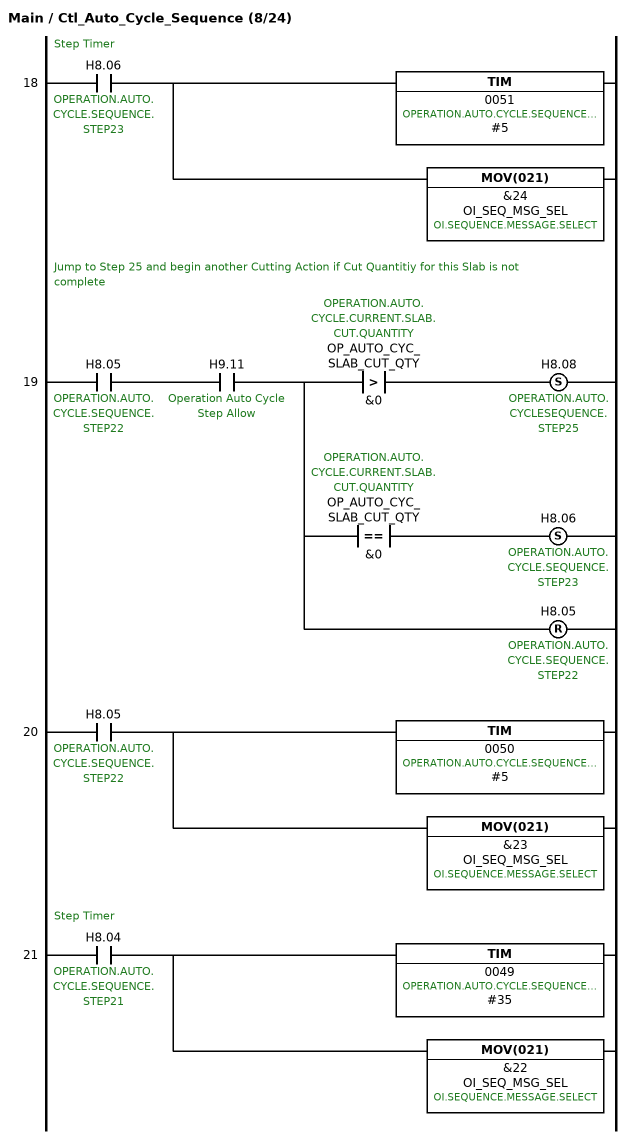
; [picture p24: Main / Ctl_Auto_Cycle_Sequence, rungs 18-21]
; rung 18: Step Timer
LD H8.06  ; OPERATION.AUTO.CYCLE.SEQUENCE.STEP23
TIM 0051 #5  ; OPERATION.AUTO.CYCLE.SEQUENCE.STEP23.TIMER
MOV(021) &24 OI_SEQ_MSG_SEL  ; OI.SEQUENCE.MESSAGE.SELECT
; rung 19: Jump to Step 25 and begin another Cutting Action if Cut Quantitiy for this Slab is not complete
LD H8.05  ; OPERATION.AUTO.CYCLE.SEQUENCE.STEP22
AND H9.11  ; Operation Auto Cycle Step Allow
OUT TR0
AND>(320) OP_AUTO_CYC_SLAB_CUT_QTY &0  ; OPERATION.AUTO.CYCLE.CURRENT.SLAB.CUT.QUANTITY
SET H8.08  ; OPERATION.AUTO.CYCLESEQUENCE.STEP25
LD TR0
AND=(300) OP_AUTO_CYC_SLAB_CUT_QTY &0  ; OPERATION.AUTO.CYCLE.CURRENT.SLAB.CUT.QUANTITY
SET H8.06  ; OPERATION.AUTO.CYCLE.SEQUENCE.STEP23
LD TR0
RSET H8.05  ; OPERATION.AUTO.CYCLE.SEQUENCE.STEP22
; rung 20
LD H8.05  ; OPERATION.AUTO.CYCLE.SEQUENCE.STEP22
TIM 0050 #5  ; OPERATION.AUTO.CYCLE.SEQUENCE.STEP22.TIMER
MOV(021) &23 OI_SEQ_MSG_SEL  ; OI.SEQUENCE.MESSAGE.SELECT
; rung 21: Step Timer
LD H8.04  ; OPERATION.AUTO.CYCLE.SEQUENCE.STEP21
TIM 0049 #35  ; OPERATION.AUTO.CYCLE.SEQUENCE.STEP21.TIMER
MOV(021) &22 OI_SEQ_MSG_SEL  ; OI.SEQUENCE.MESSAGE.SELECT

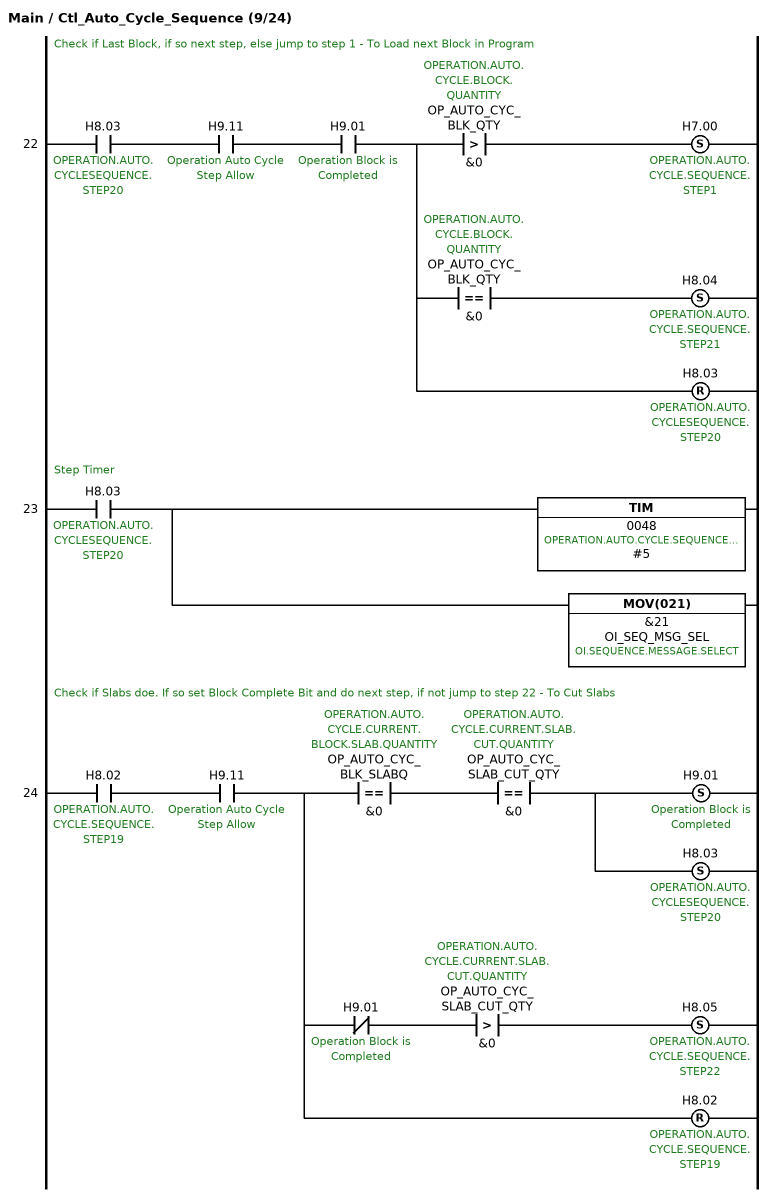
; rung 22: Check if Last Block, if so next step, else jump to step 1 - To Load next Block in Program
LD H8.03  ; OPERATION.AUTO.CYCLESEQUENCE.STEP20
AND H9.11  ; Operation Auto Cycle Step Allow
AND H9.01  ; Operation Block is Completed
OUT TR0
AND>(320) OP_AUTO_CYC_BLK_QTY &0  ; OPERATION.AUTO.CYCLE.BLOCK.QUANTITY
SET H7.00  ; OPERATION.AUTO.CYCLE.SEQUENCE.STEP1
LD TR0
AND=(300) OP_AUTO_CYC_BLK_QTY &0  ; OPERATION.AUTO.CYCLE.BLOCK.QUANTITY
SET H8.04  ; OPERATION.AUTO.CYCLE.SEQUENCE.STEP21
LD TR0
RSET H8.03  ; OPERATION.AUTO.CYCLESEQUENCE.STEP20
; rung 23: Step Timer
LD H8.03  ; OPERATION.AUTO.CYCLESEQUENCE.STEP20
TIM 0048 #5  ; OPERATION.AUTO.CYCLE.SEQUENCE.STEP20.TIMER
MOV(021) &21 OI_SEQ_MSG_SEL  ; OI.SEQUENCE.MESSAGE.SELECT
; rung 24: Check if Slabs doe. If so set Block Complete Bit and do next step, if not jump to step 22 - To Cut Slabs
LD H8.02  ; OPERATION.AUTO.CYCLE.SEQUENCE.STEP19
AND H9.11  ; Operation Auto Cycle Step Allow
OUT TR0
AND=(300) OP_AUTO_CYC_BLK_SLABQ &0  ; OPERATION.AUTO.CYCLE.CURRENT.BLOCK.SLAB.QUANTITY
AND=(300) OP_AUTO_CYC_SLAB_CUT_QTY &0  ; OPERATION.AUTO.CYCLE.CURRENT.SLAB.CUT.QUANTITY
SET H9.01  ; Operation Block is Completed
SET H8.03  ; OPERATION.AUTO.CYCLESEQUENCE.STEP20
LD TR0
ANDNOT H9.01  ; Operation Block is Completed
AND>(320) OP_AUTO_CYC_SLAB_CUT_QTY &0  ; OPERATION.AUTO.CYCLE.CURRENT.SLAB.CUT.QUANTITY
SET H8.05  ; OPERATION.AUTO.CYCLE.SEQUENCE.STEP22
LD TR0
RSET H8.02  ; OPERATION.AUTO.CYCLE.SEQUENCE.STEP19

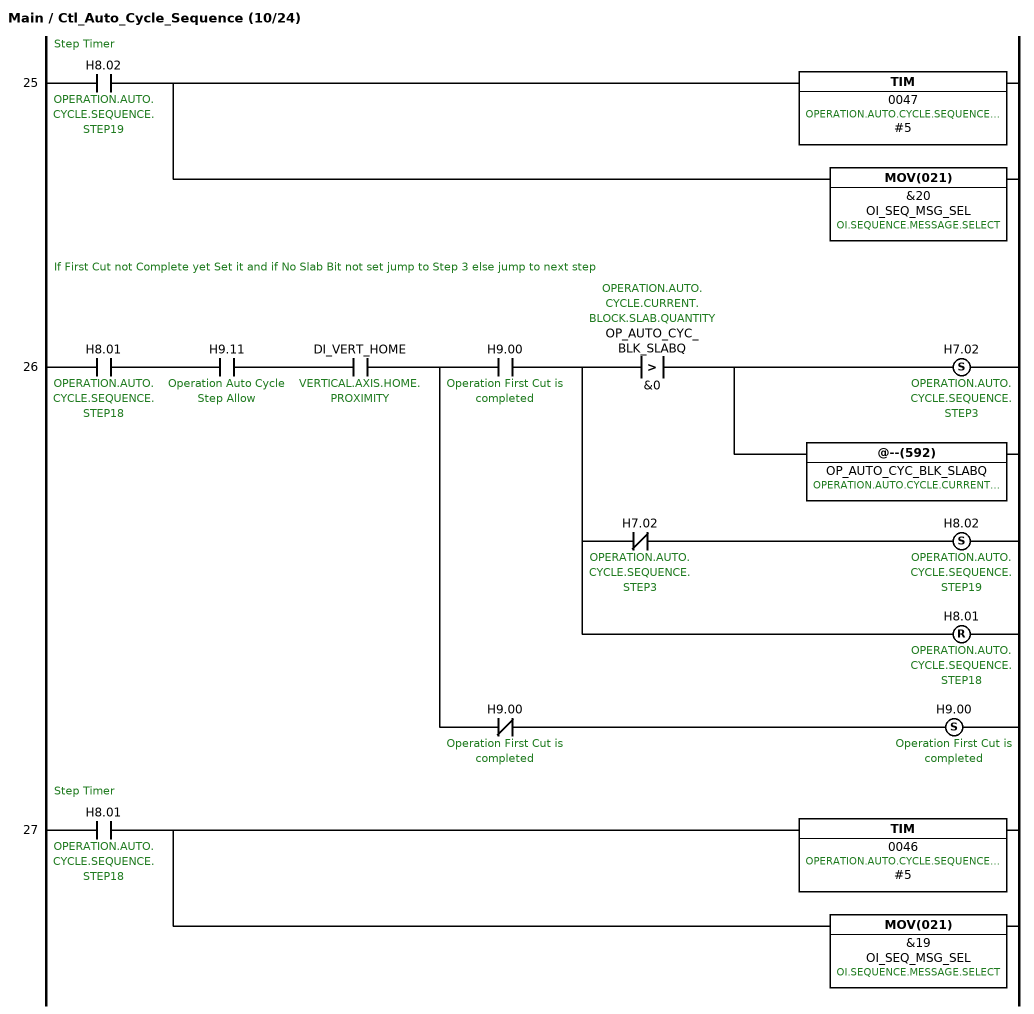
; rung 25: Step Timer
LD H8.02  ; OPERATION.AUTO.CYCLE.SEQUENCE.STEP19
TIM 0047 #5  ; OPERATION.AUTO.CYCLE.SEQUENCE.STEP19.TIMER
MOV(021) &20 OI_SEQ_MSG_SEL  ; OI.SEQUENCE.MESSAGE.SELECT
; rung 26: If First Cut not Complete yet Set it and if No Slab Bit not set jump to Step 3 else jump to next step
LD H8.01  ; OPERATION.AUTO.CYCLE.SEQUENCE.STEP18
AND H9.11  ; Operation Auto Cycle Step Allow
AND DI_VERT_HOME  ; VERTICAL.AXIS.HOME.PROXIMITY
OUT TR0
AND H9.00  ; Operation First Cut is completed
OUT TR1
AND>(320) OP_AUTO_CYC_BLK_SLABQ &0  ; OPERATION.AUTO.CYCLE.CURRENT.BLOCK.SLAB.QUANTITY
SET H7.02  ; OPERATION.AUTO.CYCLE.SEQUENCE.STEP3
@--(592) OP_AUTO_CYC_BLK_SLABQ  ; OPERATION.AUTO.CYCLE.CURRENT.BLOCK.SLAB.QUANTITY
LD TR1
ANDNOT H7.02  ; OPERATION.AUTO.CYCLE.SEQUENCE.STEP3
SET H8.02  ; OPERATION.AUTO.CYCLE.SEQUENCE.STEP19
LD TR1
RSET H8.01  ; OPERATION.AUTO.CYCLE.SEQUENCE.STEP18
LD TR0
ANDNOT H9.00  ; Operation First Cut is completed
SET H9.00  ; Operation First Cut is completed
; rung 27: Step Timer
LD H8.01  ; OPERATION.AUTO.CYCLE.SEQUENCE.STEP18
TIM 0046 #5  ; OPERATION.AUTO.CYCLE.SEQUENCE.STEP18.TIMER
MOV(021) &19 OI_SEQ_MSG_SEL  ; OI.SEQUENCE.MESSAGE.SELECT

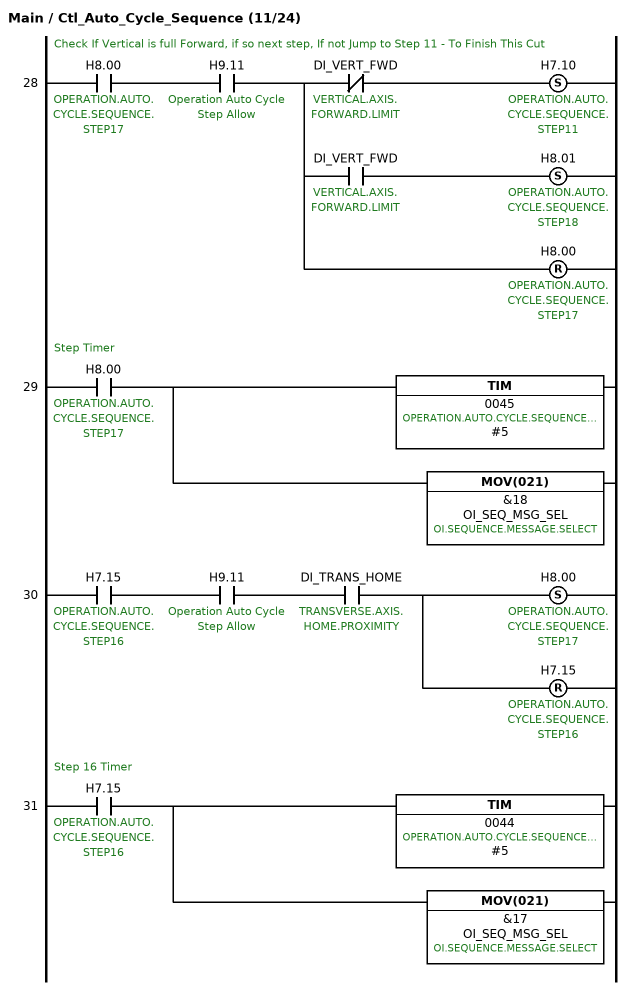
; rung 28: Check If Vertical is full Forward, if so next step, If not Jump to Step 11 - To Finish This Cut
LD H8.00  ; OPERATION.AUTO.CYCLE.SEQUENCE.STEP17
AND H9.11  ; Operation Auto Cycle Step Allow
OUT TR0
ANDNOT DI_VERT_FWD  ; VERTICAL.AXIS.FORWARD.LIMIT
SET H7.10  ; OPERATION.AUTO.CYCLE.SEQUENCE.STEP11
LD TR0
AND DI_VERT_FWD  ; VERTICAL.AXIS.FORWARD.LIMIT
SET H8.01  ; OPERATION.AUTO.CYCLE.SEQUENCE.STEP18
LD TR0
RSET H8.00  ; OPERATION.AUTO.CYCLE.SEQUENCE.STEP17
; rung 29: Step Timer
LD H8.00  ; OPERATION.AUTO.CYCLE.SEQUENCE.STEP17
TIM 0045 #5  ; OPERATION.AUTO.CYCLE.SEQUENCE.STEP17.TIMER
MOV(021) &18 OI_SEQ_MSG_SEL  ; OI.SEQUENCE.MESSAGE.SELECT
; rung 30
LD H7.15  ; OPERATION.AUTO.CYCLE.SEQUENCE.STEP16
AND H9.11  ; Operation Auto Cycle Step Allow
AND DI_TRANS_HOME  ; TRANSVERSE.AXIS.HOME.PROXIMITY
SET H8.00  ; OPERATION.AUTO.CYCLE.SEQUENCE.STEP17
RSET H7.15  ; OPERATION.AUTO.CYCLE.SEQUENCE.STEP16
; rung 31: Step 16 Timer
LD H7.15  ; OPERATION.AUTO.CYCLE.SEQUENCE.STEP16
TIM 0044 #5  ; OPERATION.AUTO.CYCLE.SEQUENCE.STEP16.TIMER
MOV(021) &17 OI_SEQ_MSG_SEL  ; OI.SEQUENCE.MESSAGE.SELECT

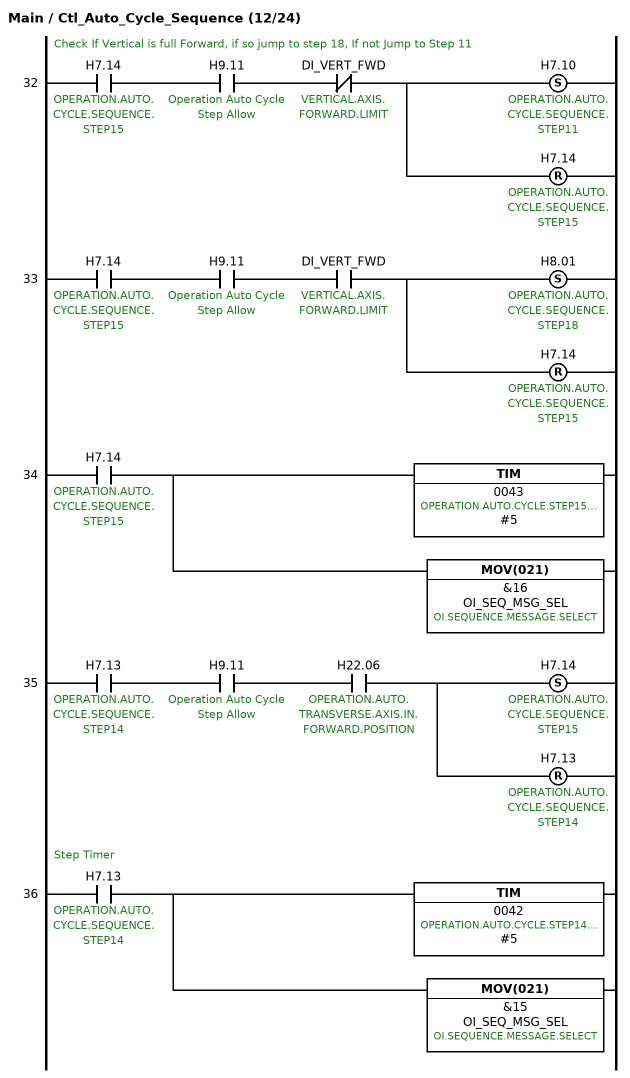
; rung 32: Check If Vertical is full Forward, if so jump to step 18, If not Jump to Step 11
LD H7.14  ; OPERATION.AUTO.CYCLE.SEQUENCE.STEP15
AND H9.11  ; Operation Auto Cycle Step Allow
ANDNOT DI_VERT_FWD  ; VERTICAL.AXIS.FORWARD.LIMIT
SET H7.10  ; OPERATION.AUTO.CYCLE.SEQUENCE.STEP11
RSET H7.14  ; OPERATION.AUTO.CYCLE.SEQUENCE.STEP15
; rung 33
LD H7.14  ; OPERATION.AUTO.CYCLE.SEQUENCE.STEP15
AND H9.11  ; Operation Auto Cycle Step Allow
AND DI_VERT_FWD  ; VERTICAL.AXIS.FORWARD.LIMIT
SET H8.01  ; OPERATION.AUTO.CYCLE.SEQUENCE.STEP18
RSET H7.14  ; OPERATION.AUTO.CYCLE.SEQUENCE.STEP15
; rung 34
LD H7.14  ; OPERATION.AUTO.CYCLE.SEQUENCE.STEP15
TIM 0043 #5  ; OPERATION.AUTO.CYCLE.STEP15.TIMER
MOV(021) &16 OI_SEQ_MSG_SEL  ; OI.SEQUENCE.MESSAGE.SELECT
; rung 35
LD H7.13  ; OPERATION.AUTO.CYCLE.SEQUENCE.STEP14
AND H9.11  ; Operation Auto Cycle Step Allow
AND H22.06  ; OPERATION.AUTO.TRANSVERSE.AXIS.IN.FORWARD.POSITION
SET H7.14  ; OPERATION.AUTO.CYCLE.SEQUENCE.STEP15
RSET H7.13  ; OPERATION.AUTO.CYCLE.SEQUENCE.STEP14
; rung 36: Step Timer
LD H7.13  ; OPERATION.AUTO.CYCLE.SEQUENCE.STEP14
TIM 0042 #5  ; OPERATION.AUTO.CYCLE.STEP14.TIMER
MOV(021) &15 OI_SEQ_MSG_SEL  ; OI.SEQUENCE.MESSAGE.SELECT

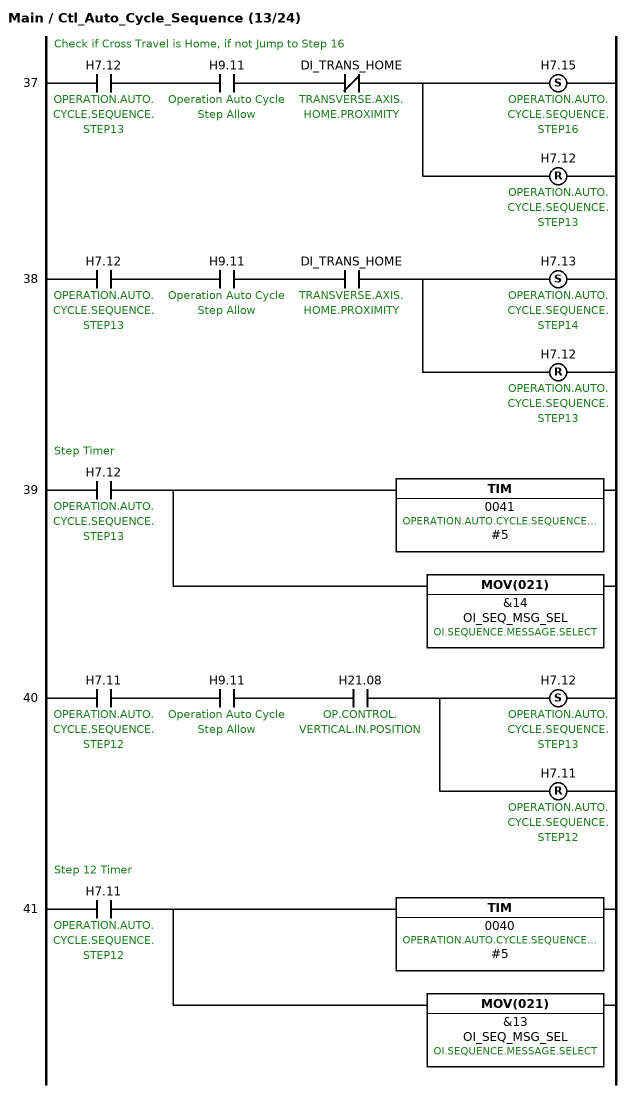
; rung 37: Check if Cross Travel is Home, if not Jump to Step 16
LD H7.12  ; OPERATION.AUTO.CYCLE.SEQUENCE.STEP13
AND H9.11  ; Operation Auto Cycle Step Allow
ANDNOT DI_TRANS_HOME  ; TRANSVERSE.AXIS.HOME.PROXIMITY
SET H7.15  ; OPERATION.AUTO.CYCLE.SEQUENCE.STEP16
RSET H7.12  ; OPERATION.AUTO.CYCLE.SEQUENCE.STEP13
; rung 38
LD H7.12  ; OPERATION.AUTO.CYCLE.SEQUENCE.STEP13
AND H9.11  ; Operation Auto Cycle Step Allow
AND DI_TRANS_HOME  ; TRANSVERSE.AXIS.HOME.PROXIMITY
SET H7.13  ; OPERATION.AUTO.CYCLE.SEQUENCE.STEP14
RSET H7.12  ; OPERATION.AUTO.CYCLE.SEQUENCE.STEP13
; rung 39: Step Timer
LD H7.12  ; OPERATION.AUTO.CYCLE.SEQUENCE.STEP13
TIM 0041 #5  ; OPERATION.AUTO.CYCLE.SEQUENCE.STEP13.TIME
MOV(021) &14 OI_SEQ_MSG_SEL  ; OI.SEQUENCE.MESSAGE.SELECT
; rung 40
LD H7.11  ; OPERATION.AUTO.CYCLE.SEQUENCE.STEP12
AND H9.11  ; Operation Auto Cycle Step Allow
AND H21.08  ; OP.CONTROL.VERTICAL.IN.POSITION
SET H7.12  ; OPERATION.AUTO.CYCLE.SEQUENCE.STEP13
RSET H7.11  ; OPERATION.AUTO.CYCLE.SEQUENCE.STEP12
; rung 41: Step 12 Timer
LD H7.11  ; OPERATION.AUTO.CYCLE.SEQUENCE.STEP12
TIM 0040 #5  ; OPERATION.AUTO.CYCLE.SEQUENCE.STEP12.TIMER
MOV(021) &13 OI_SEQ_MSG_SEL  ; OI.SEQUENCE.MESSAGE.SELECT

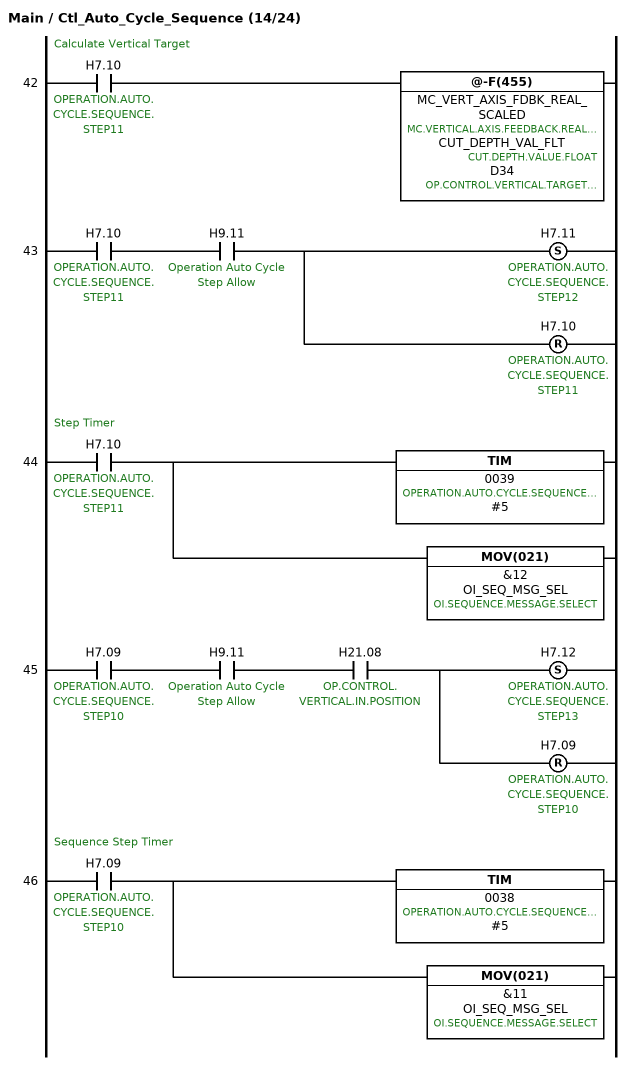
; rung 42: Calculate Vertical Target
LD H7.10  ; OPERATION.AUTO.CYCLE.SEQUENCE.STEP11
@-F(455) MC_VERT_AXIS_FDBK_REAL_SCALED CUT_DEPTH_VAL_FLT D34  ; MC.VERTICAL.AXIS.FEEDBACK.REAL.SCALED.INCH, CUT.DEPTH.VALUE.FLOAT, OP.CONTROL.VERTICAL.TARGET.SCALED
; rung 43
LD H7.10  ; OPERATION.AUTO.CYCLE.SEQUENCE.STEP11
AND H9.11  ; Operation Auto Cycle Step Allow
SET H7.11  ; OPERATION.AUTO.CYCLE.SEQUENCE.STEP12
RSET H7.10  ; OPERATION.AUTO.CYCLE.SEQUENCE.STEP11
; rung 44: Step Timer
LD H7.10  ; OPERATION.AUTO.CYCLE.SEQUENCE.STEP11
TIM 0039 #5  ; OPERATION.AUTO.CYCLE.SEQUENCE.STEP11.TIMER
MOV(021) &12 OI_SEQ_MSG_SEL  ; OI.SEQUENCE.MESSAGE.SELECT
; rung 45
LD H7.09  ; OPERATION.AUTO.CYCLE.SEQUENCE.STEP10
AND H9.11  ; Operation Auto Cycle Step Allow
AND H21.08  ; OP.CONTROL.VERTICAL.IN.POSITION
SET H7.12  ; OPERATION.AUTO.CYCLE.SEQUENCE.STEP13
RSET H7.09  ; OPERATION.AUTO.CYCLE.SEQUENCE.STEP10
; rung 46: Sequence Step Timer
LD H7.09  ; OPERATION.AUTO.CYCLE.SEQUENCE.STEP10
TIM 0038 #5  ; OPERATION.AUTO.CYCLE.SEQUENCE.STEP10.TIMER
MOV(021) &11 OI_SEQ_MSG_SEL  ; OI.SEQUENCE.MESSAGE.SELECT

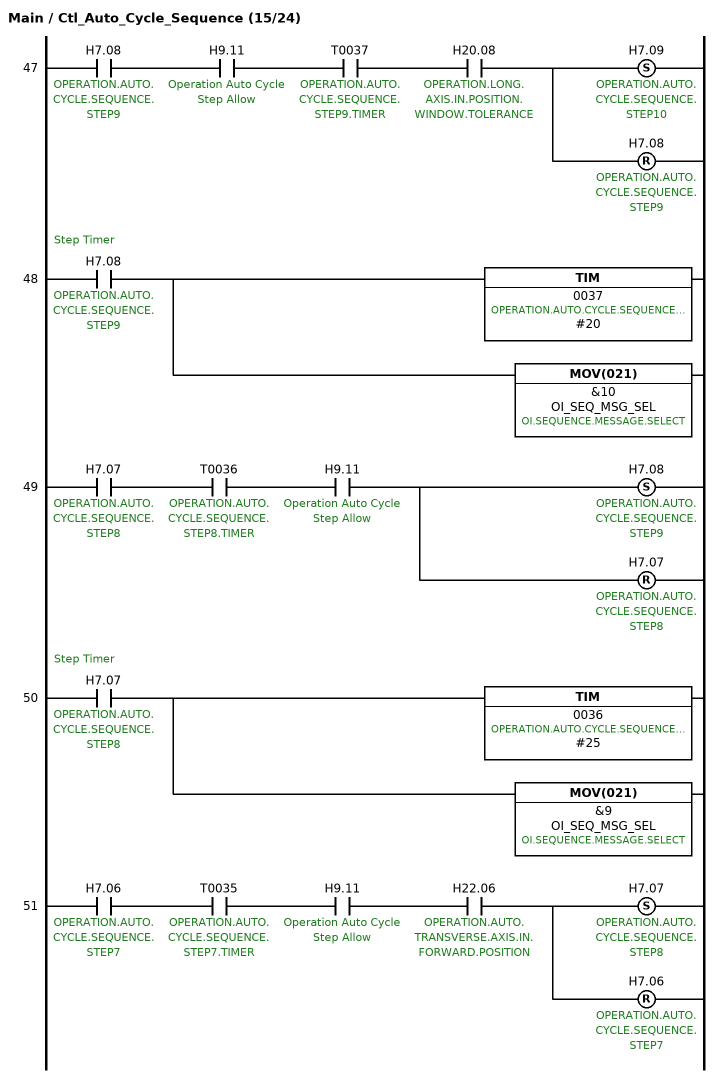
; rung 47
LD H7.08  ; OPERATION.AUTO.CYCLE.SEQUENCE.STEP9
AND H9.11  ; Operation Auto Cycle Step Allow
AND T0037  ; OPERATION.AUTO.CYCLE.SEQUENCE.STEP9.TIMER
AND H20.08  ; OPERATION.LONG.AXIS.IN.POSITION.WINDOW.TOLERANCE
SET H7.09  ; OPERATION.AUTO.CYCLE.SEQUENCE.STEP10
RSET H7.08  ; OPERATION.AUTO.CYCLE.SEQUENCE.STEP9
; rung 48: Step Timer
LD H7.08  ; OPERATION.AUTO.CYCLE.SEQUENCE.STEP9
TIM 0037 #20  ; OPERATION.AUTO.CYCLE.SEQUENCE.STEP9.TIMER
MOV(021) &10 OI_SEQ_MSG_SEL  ; OI.SEQUENCE.MESSAGE.SELECT
; rung 49
LD H7.07  ; OPERATION.AUTO.CYCLE.SEQUENCE.STEP8
AND T0036  ; OPERATION.AUTO.CYCLE.SEQUENCE.STEP8.TIMER
AND H9.11  ; Operation Auto Cycle Step Allow
SET H7.08  ; OPERATION.AUTO.CYCLE.SEQUENCE.STEP9
RSET H7.07  ; OPERATION.AUTO.CYCLE.SEQUENCE.STEP8
; rung 50: Step Timer
LD H7.07  ; OPERATION.AUTO.CYCLE.SEQUENCE.STEP8
TIM 0036 #25  ; OPERATION.AUTO.CYCLE.SEQUENCE.STEP8.TIMER
MOV(021) &9 OI_SEQ_MSG_SEL  ; OI.SEQUENCE.MESSAGE.SELECT
; rung 51
LD H7.06  ; OPERATION.AUTO.CYCLE.SEQUENCE.STEP7
AND T0035  ; OPERATION.AUTO.CYCLE.SEQUENCE.STEP7.TIMER
AND H9.11  ; Operation Auto Cycle Step Allow
AND H22.06  ; OPERATION.AUTO.TRANSVERSE.AXIS.IN.FORWARD.POSITION
SET H7.07  ; OPERATION.AUTO.CYCLE.SEQUENCE.STEP8
RSET H7.06  ; OPERATION.AUTO.CYCLE.SEQUENCE.STEP7

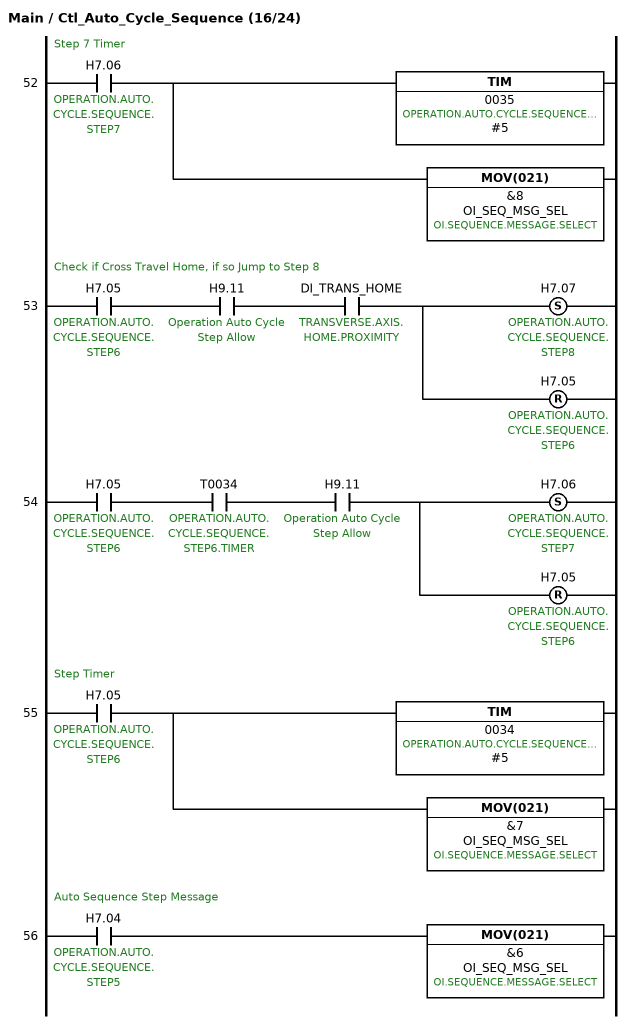
; rung 52: Step 7 Timer
LD H7.06  ; OPERATION.AUTO.CYCLE.SEQUENCE.STEP7
TIM 0035 #5  ; OPERATION.AUTO.CYCLE.SEQUENCE.STEP7.TIMER
MOV(021) &8 OI_SEQ_MSG_SEL  ; OI.SEQUENCE.MESSAGE.SELECT
; rung 53: Check if Cross Travel Home, if so Jump to Step 8
LD H7.05  ; OPERATION.AUTO.CYCLE.SEQUENCE.STEP6
AND H9.11  ; Operation Auto Cycle Step Allow
AND DI_TRANS_HOME  ; TRANSVERSE.AXIS.HOME.PROXIMITY
SET H7.07  ; OPERATION.AUTO.CYCLE.SEQUENCE.STEP8
RSET H7.05  ; OPERATION.AUTO.CYCLE.SEQUENCE.STEP6
; rung 54
LD H7.05  ; OPERATION.AUTO.CYCLE.SEQUENCE.STEP6
AND T0034  ; OPERATION.AUTO.CYCLE.SEQUENCE.STEP6.TIMER
AND H9.11  ; Operation Auto Cycle Step Allow
SET H7.06  ; OPERATION.AUTO.CYCLE.SEQUENCE.STEP7
RSET H7.05  ; OPERATION.AUTO.CYCLE.SEQUENCE.STEP6
; rung 55: Step Timer
LD H7.05  ; OPERATION.AUTO.CYCLE.SEQUENCE.STEP6
TIM 0034 #5  ; OPERATION.AUTO.CYCLE.SEQUENCE.STEP6.TIMER
MOV(021) &7 OI_SEQ_MSG_SEL  ; OI.SEQUENCE.MESSAGE.SELECT
; rung 56: Auto Sequence Step Message
LD H7.04  ; OPERATION.AUTO.CYCLE.SEQUENCE.STEP5
MOV(021) &6 OI_SEQ_MSG_SEL  ; OI.SEQUENCE.MESSAGE.SELECT

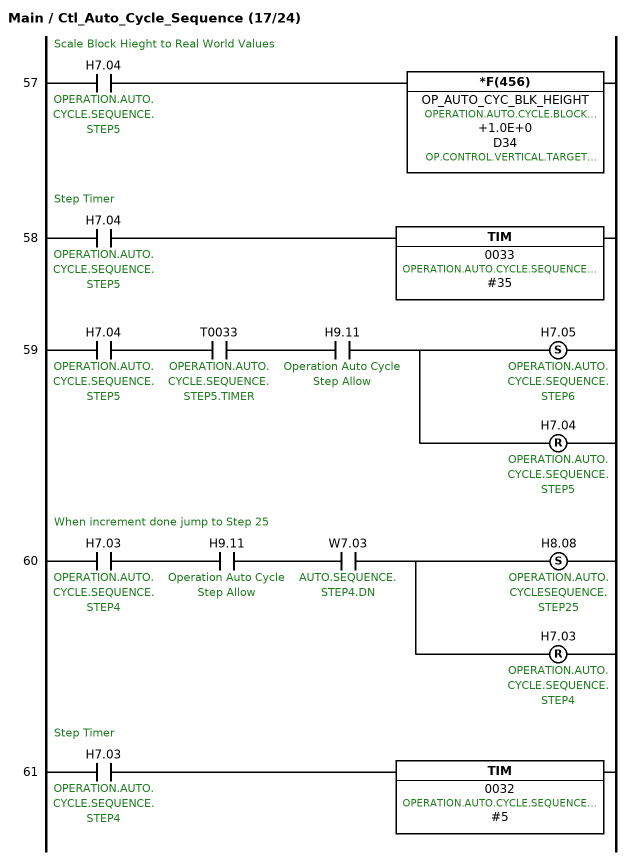
; rung 57: Scale Block Hieght to Real World Values
LD H7.04  ; OPERATION.AUTO.CYCLE.SEQUENCE.STEP5
*F(456) OP_AUTO_CYC_BLK_HEIGHT +1.0E+0 D34  ; OPERATION.AUTO.CYCLE.BLOCK.HEIGHT.WORKING, OP.CONTROL.VERTICAL.TARGET.SCALED
; rung 58: Step Timer
LD H7.04  ; OPERATION.AUTO.CYCLE.SEQUENCE.STEP5
TIM 0033 #35  ; OPERATION.AUTO.CYCLE.SEQUENCE.STEP5.TIMER
; rung 59
LD H7.04  ; OPERATION.AUTO.CYCLE.SEQUENCE.STEP5
AND T0033  ; OPERATION.AUTO.CYCLE.SEQUENCE.STEP5.TIMER
AND H9.11  ; Operation Auto Cycle Step Allow
SET H7.05  ; OPERATION.AUTO.CYCLE.SEQUENCE.STEP6
RSET H7.04  ; OPERATION.AUTO.CYCLE.SEQUENCE.STEP5
; rung 60: When increment done jump to Step 25
LD H7.03  ; OPERATION.AUTO.CYCLE.SEQUENCE.STEP4
AND H9.11  ; Operation Auto Cycle Step Allow
AND W7.03  ; AUTO.SEQUENCE.STEP4.DN
SET H8.08  ; OPERATION.AUTO.CYCLESEQUENCE.STEP25
RSET H7.03  ; OPERATION.AUTO.CYCLE.SEQUENCE.STEP4
; rung 61: Step Timer
LD H7.03  ; OPERATION.AUTO.CYCLE.SEQUENCE.STEP4
TIM 0032 #5  ; OPERATION.AUTO.CYCLE.SEQUENCE.STEP4.TIMER

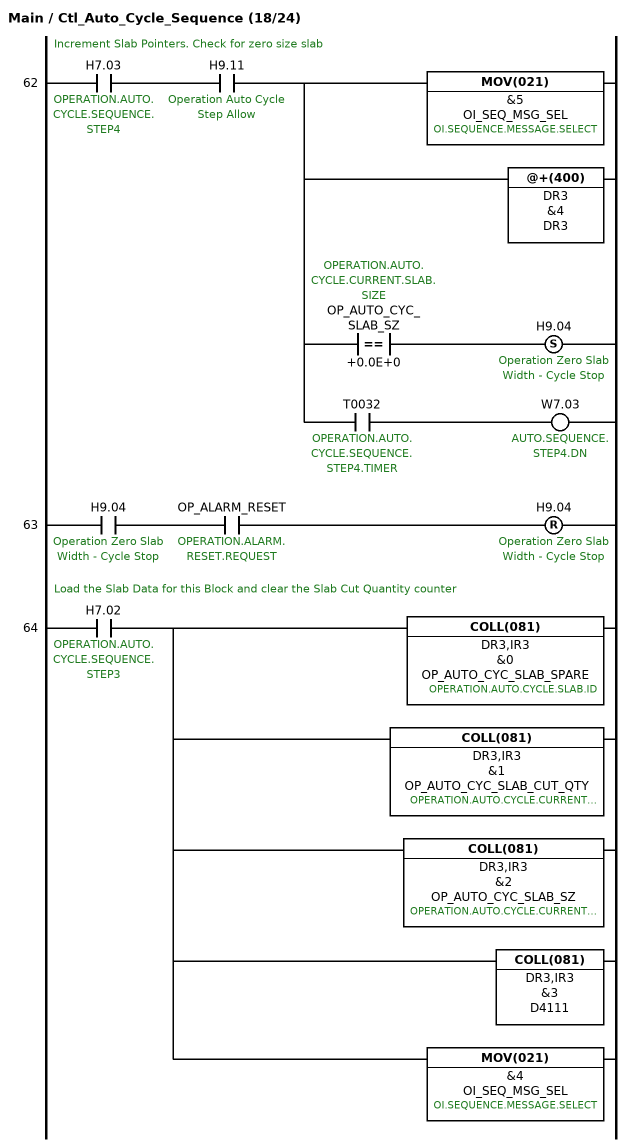
; rung 62: Increment Slab Pointers. Check for zero size slab
LD H7.03  ; OPERATION.AUTO.CYCLE.SEQUENCE.STEP4
AND H9.11  ; Operation Auto Cycle Step Allow
OUT TR0
MOV(021) &5 OI_SEQ_MSG_SEL  ; OI.SEQUENCE.MESSAGE.SELECT
@+(400) DR3 &4 DR3
AND=F(329) OP_AUTO_CYC_SLAB_SZ +0.0E+0  ; OPERATION.AUTO.CYCLE.CURRENT.SLAB.SIZE
SET H9.04  ; Operation Zero Slab Width - Cycle Stop
LD TR0
AND T0032  ; OPERATION.AUTO.CYCLE.SEQUENCE.STEP4.TIMER
OUT W7.03  ; AUTO.SEQUENCE.STEP4.DN
; rung 63
LD H9.04  ; Operation Zero Slab Width - Cycle Stop
AND OP_ALARM_RESET  ; OPERATION.ALARM.RESET.REQUEST
RSET H9.04  ; Operation Zero Slab Width - Cycle Stop
; rung 64: Load the Slab Data for this Block and clear the Slab Cut Quantity counter
LD H7.02  ; OPERATION.AUTO.CYCLE.SEQUENCE.STEP3
COLL(081) DR3,IR3 &0 OP_AUTO_CYC_SLAB_SPARE  ; OPERATION.AUTO.CYCLE.SLAB.ID
COLL(081) DR3,IR3 &1 OP_AUTO_CYC_SLAB_CUT_QTY  ; OPERATION.AUTO.CYCLE.CURRENT.SLAB.CUT.QUANTITY
COLL(081) DR3,IR3 &2 OP_AUTO_CYC_SLAB_SZ  ; OPERATION.AUTO.CYCLE.CURRENT.SLAB.SIZE
COLL(081) DR3,IR3 &3 D4111
MOV(021) &4 OI_SEQ_MSG_SEL  ; OI.SEQUENCE.MESSAGE.SELECT

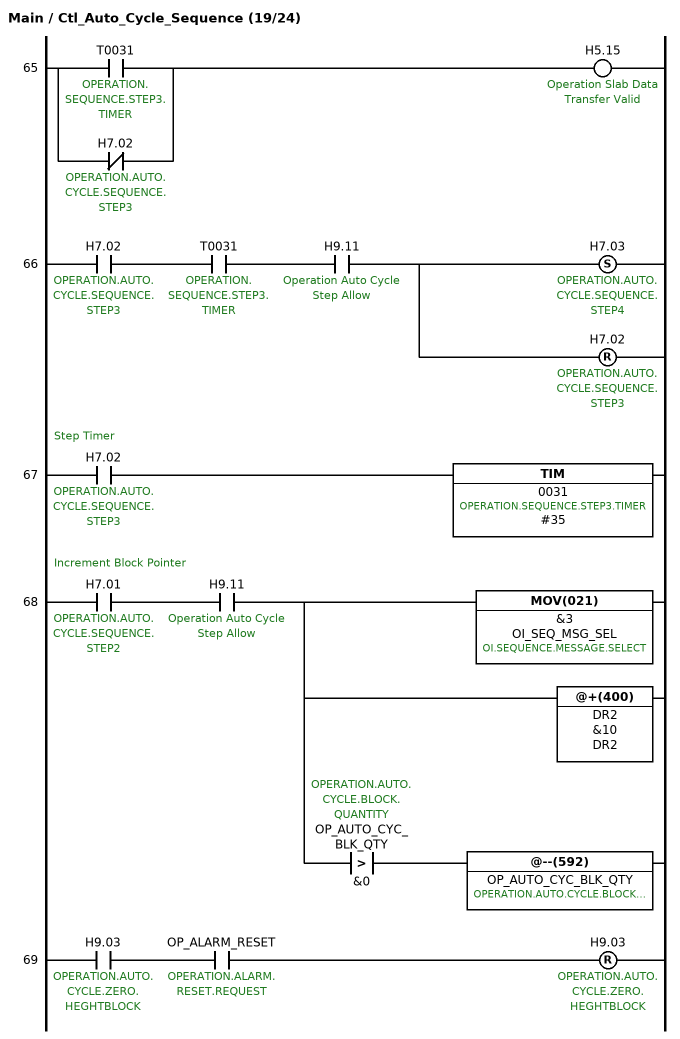
; rung 65
LD T0031  ; OPERATION.SEQUENCE.STEP3.TIMER
ORNOT H7.02  ; OPERATION.AUTO.CYCLE.SEQUENCE.STEP3
OUT H5.15  ; Operation Slab Data Transfer Valid
; rung 66
LD H7.02  ; OPERATION.AUTO.CYCLE.SEQUENCE.STEP3
AND T0031  ; OPERATION.SEQUENCE.STEP3.TIMER
AND H9.11  ; Operation Auto Cycle Step Allow
SET H7.03  ; OPERATION.AUTO.CYCLE.SEQUENCE.STEP4
RSET H7.02  ; OPERATION.AUTO.CYCLE.SEQUENCE.STEP3
; rung 67: Step Timer
LD H7.02  ; OPERATION.AUTO.CYCLE.SEQUENCE.STEP3
TIM 0031 #35  ; OPERATION.SEQUENCE.STEP3.TIMER
; rung 68: Increment Block Pointer
LD H7.01  ; OPERATION.AUTO.CYCLE.SEQUENCE.STEP2
AND H9.11  ; Operation Auto Cycle Step Allow
MOV(021) &3 OI_SEQ_MSG_SEL  ; OI.SEQUENCE.MESSAGE.SELECT
@+(400) DR2 &10 DR2
AND>(320) OP_AUTO_CYC_BLK_QTY &0  ; OPERATION.AUTO.CYCLE.BLOCK.QUANTITY
@--(592) OP_AUTO_CYC_BLK_QTY  ; OPERATION.AUTO.CYCLE.BLOCK.QUANTITY
; rung 69
LD H9.03  ; OPERATION.AUTO.CYCLE.ZERO.HEGHTBLOCK
AND OP_ALARM_RESET  ; OPERATION.ALARM.RESET.REQUEST
RSET H9.03  ; OPERATION.AUTO.CYCLE.ZERO.HEGHTBLOCK

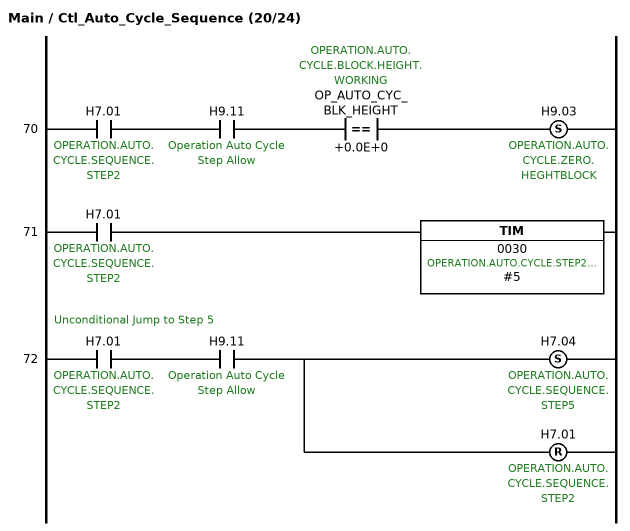
; rung 70
LD H7.01  ; OPERATION.AUTO.CYCLE.SEQUENCE.STEP2
AND H9.11  ; Operation Auto Cycle Step Allow
AND=F(329) OP_AUTO_CYC_BLK_HEIGHT +0.0E+0  ; OPERATION.AUTO.CYCLE.BLOCK.HEIGHT.WORKING
SET H9.03  ; OPERATION.AUTO.CYCLE.ZERO.HEGHTBLOCK
; rung 71
LD H7.01  ; OPERATION.AUTO.CYCLE.SEQUENCE.STEP2
TIM 0030 #5  ; OPERATION.AUTO.CYCLE.STEP2.TIMER
; rung 72: Unconditional Jump to Step 5
LD H7.01  ; OPERATION.AUTO.CYCLE.SEQUENCE.STEP2
AND H9.11  ; Operation Auto Cycle Step Allow
SET H7.04  ; OPERATION.AUTO.CYCLE.SEQUENCE.STEP5
RSET H7.01  ; OPERATION.AUTO.CYCLE.SEQUENCE.STEP2

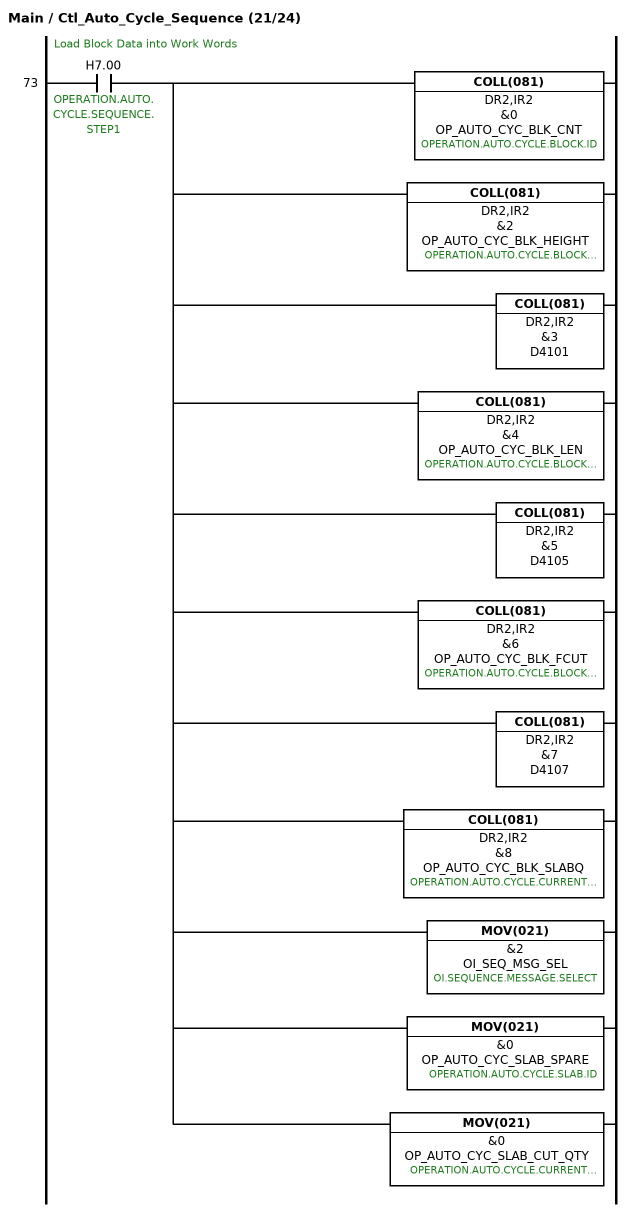
; rung 73: Load Block Data into Work Words
LD H7.00  ; OPERATION.AUTO.CYCLE.SEQUENCE.STEP1
COLL(081) DR2,IR2 &0 OP_AUTO_CYC_BLK_CNT  ; OPERATION.AUTO.CYCLE.BLOCK.ID
COLL(081) DR2,IR2 &2 OP_AUTO_CYC_BLK_HEIGHT  ; OPERATION.AUTO.CYCLE.BLOCK.HEIGHT.WORKING
COLL(081) DR2,IR2 &3 D4101
COLL(081) DR2,IR2 &4 OP_AUTO_CYC_BLK_LEN  ; OPERATION.AUTO.CYCLE.BLOCK.TRANSVERSE.AXIS.STOP.POSITION.WORKING
COLL(081) DR2,IR2 &5 D4105
COLL(081) DR2,IR2 &6 OP_AUTO_CYC_BLK_FCUT  ; OPERATION.AUTO.CYCLE.BLOCK.FIRST.CUT.WORKING
COLL(081) DR2,IR2 &7 D4107
COLL(081) DR2,IR2 &8 OP_AUTO_CYC_BLK_SLABQ  ; OPERATION.AUTO.CYCLE.CURRENT.BLOCK.SLAB.QUANTITY
MOV(021) &2 OI_SEQ_MSG_SEL  ; OI.SEQUENCE.MESSAGE.SELECT
MOV(021) &0 OP_AUTO_CYC_SLAB_SPARE  ; OPERATION.AUTO.CYCLE.SLAB.ID
MOV(021) &0 OP_AUTO_CYC_SLAB_CUT_QTY  ; OPERATION.AUTO.CYCLE.CURRENT.SLAB.CUT.QUANTITY

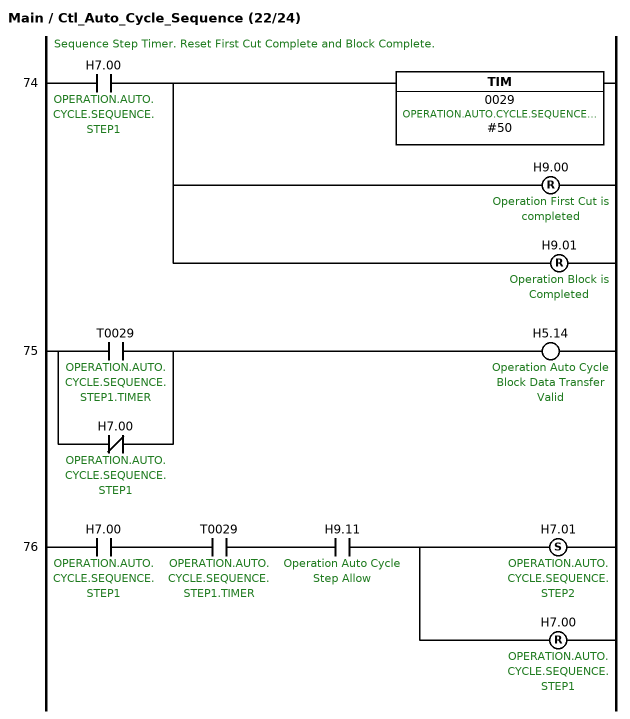
; rung 74: Sequence Step Timer. Reset First Cut Complete and Block Complete.
LD H7.00  ; OPERATION.AUTO.CYCLE.SEQUENCE.STEP1
TIM 0029 #50  ; OPERATION.AUTO.CYCLE.SEQUENCE.STEP1.TIMER
RSET H9.00  ; Operation First Cut is completed
RSET H9.01  ; Operation Block is Completed
; rung 75
LD T0029  ; OPERATION.AUTO.CYCLE.SEQUENCE.STEP1.TIMER
ORNOT H7.00  ; OPERATION.AUTO.CYCLE.SEQUENCE.STEP1
OUT H5.14  ; Operation Auto Cycle Block Data Transfer Valid
; rung 76
LD H7.00  ; OPERATION.AUTO.CYCLE.SEQUENCE.STEP1
AND T0029  ; OPERATION.AUTO.CYCLE.SEQUENCE.STEP1.TIMER
AND H9.11  ; Operation Auto Cycle Step Allow
SET H7.01  ; OPERATION.AUTO.CYCLE.SEQUENCE.STEP2
RSET H7.00  ; OPERATION.AUTO.CYCLE.SEQUENCE.STEP1

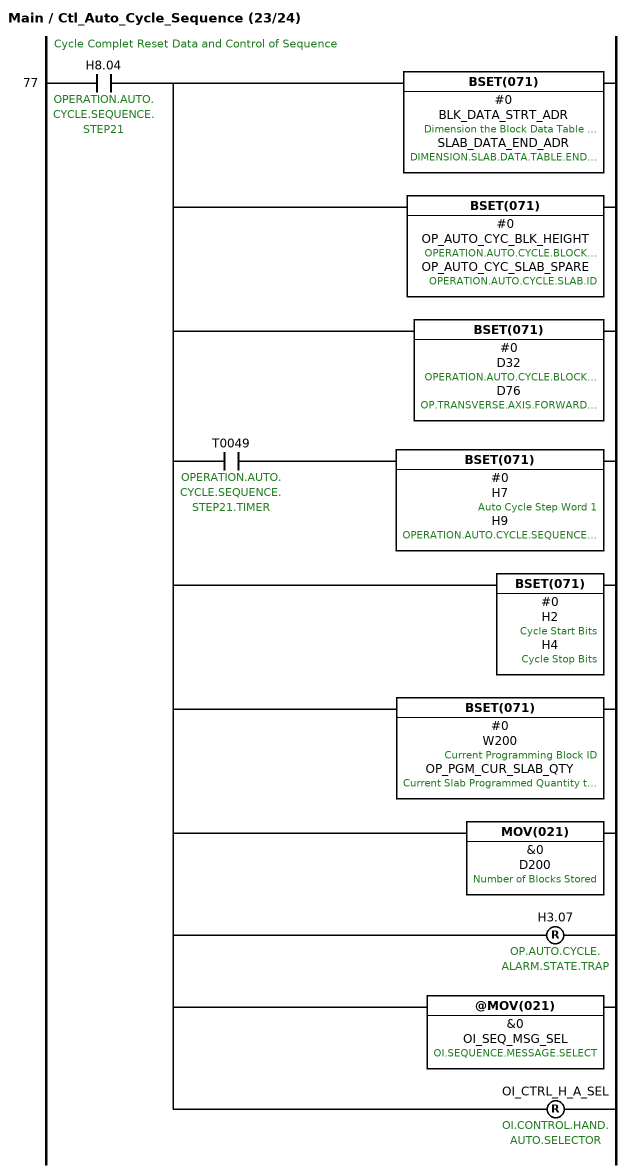
; rung 77: Cycle Complet Reset Data and Control of Sequence
LD H8.04  ; OPERATION.AUTO.CYCLE.SEQUENCE.STEP21
OUT TR0
BSET(071) #0 BLK_DATA_STRT_ADR SLAB_DATA_END_ADR  ; Dimension the Block Data Table - Start Address, DIMENSION.SLAB.DATA.TABLE.END.ADDRESS
BSET(071) #0 OP_AUTO_CYC_BLK_HEIGHT OP_AUTO_CYC_SLAB_SPARE  ; OPERATION.AUTO.CYCLE.BLOCK.HEIGHT.WORKING, OPERATION.AUTO.CYCLE.SLAB.ID
BSET(071) #0 D32 D76  ; OPERATION.AUTO.CYCLE.BLOCK.FIRST.CUT.WORKING.REAL, OP.TRANSVERSE.AXIS.FORWARD.TARGET
AND T0049  ; OPERATION.AUTO.CYCLE.SEQUENCE.STEP21.TIMER
BSET(071) #0 H7 H9  ; Auto Cycle Step Word 1, OPERATION.AUTO.CYCLE.SEQUENCE.STATE.BITS
LD TR0
BSET(071) #0 H2 H4  ; Cycle Start Bits, Cycle Stop Bits
BSET(071) #0 W200 OP_PGM_CUR_SLAB_QTY  ; Current Programming Block ID, Current Slab Programmed Quantity to cut
MOV(021) &0 D200  ; Number of Blocks Stored
RSET H3.07  ; OP.AUTO.CYCLE.ALARM.STATE.TRAP
@MOV(021) &0 OI_SEQ_MSG_SEL  ; OI.SEQUENCE.MESSAGE.SELECT
RSET OI_CTRL_H_A_SEL  ; OI.CONTROL.HAND.AUTO.SELECTOR

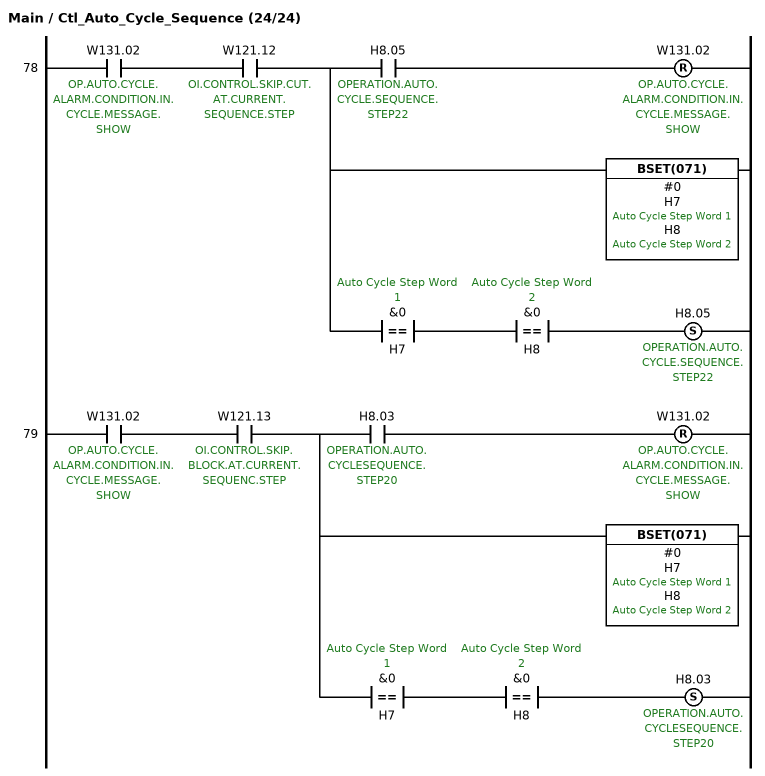
; rung 78
LD W131.02  ; OP.AUTO.CYCLE.ALARM.CONDITION.IN.CYCLE.MESSAGE.SHOW
AND W121.12  ; OI.CONTROL.SKIP.CUT.AT.CURRENT.SEQUENCE.STEP
OUT TR0
AND H8.05  ; OPERATION.AUTO.CYCLE.SEQUENCE.STEP22
RSET W131.02  ; OP.AUTO.CYCLE.ALARM.CONDITION.IN.CYCLE.MESSAGE.SHOW
LD TR0
BSET(071) #0 H7 H8  ; Auto Cycle Step Word 1, Auto Cycle Step Word 2
AND=(300) &0 H7  ; Auto Cycle Step Word 1
AND=(300) &0 H8  ; Auto Cycle Step Word 2
SET H8.05  ; OPERATION.AUTO.CYCLE.SEQUENCE.STEP22
; rung 79
LD W131.02  ; OP.AUTO.CYCLE.ALARM.CONDITION.IN.CYCLE.MESSAGE.SHOW
AND W121.13  ; OI.CONTROL.SKIP.BLOCK.AT.CURRENT.SEQUENC.STEP
OUT TR0
AND H8.03  ; OPERATION.AUTO.CYCLESEQUENCE.STEP20
RSET W131.02  ; OP.AUTO.CYCLE.ALARM.CONDITION.IN.CYCLE.MESSAGE.SHOW
LD TR0
BSET(071) #0 H7 H8  ; Auto Cycle Step Word 1, Auto Cycle Step Word 2
AND=(300) &0 H7  ; Auto Cycle Step Word 1
AND=(300) &0 H8  ; Auto Cycle Step Word 2
SET H8.03  ; OPERATION.AUTO.CYCLESEQUENCE.STEP20

### Section Ctl_Master_Home

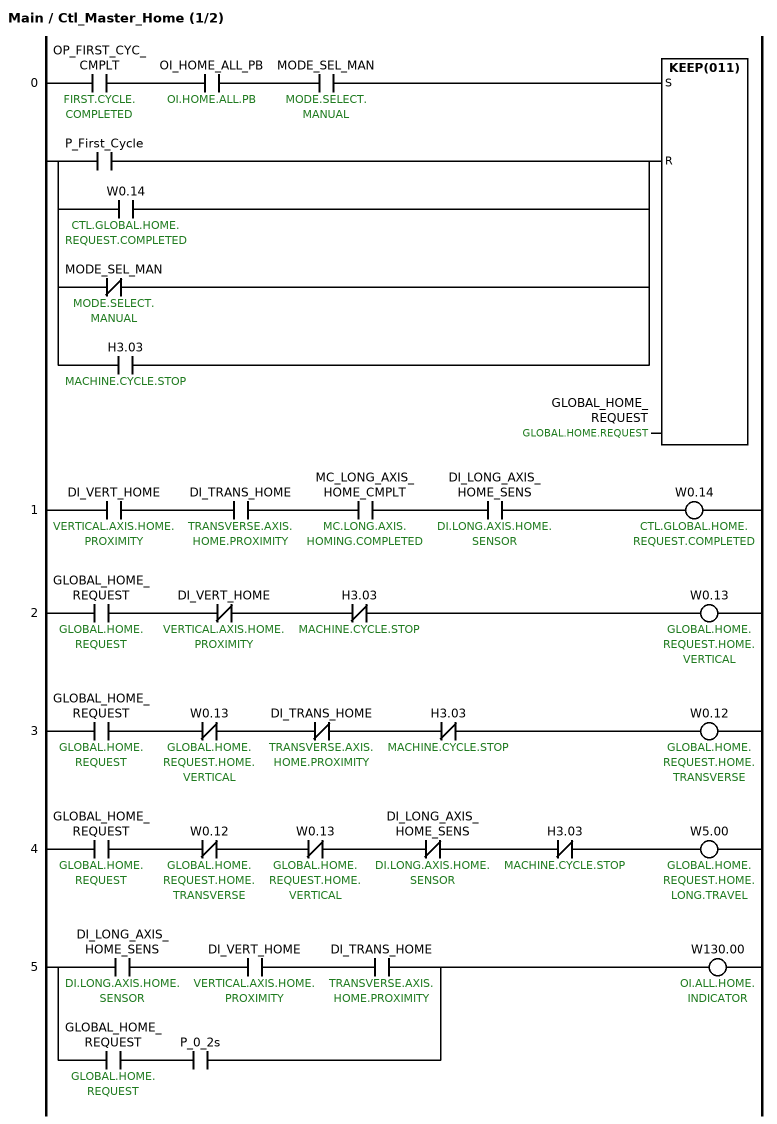
; rung 0
LD OP_FIRST_CYC_CMPLT  ; FIRST.CYCLE.COMPLETED
AND OI_HOME_ALL_PB  ; OI.HOME.ALL.PB
AND MODE_SEL_MAN  ; MODE.SELECT.MANUAL
LD P_First_Cycle
OR W0.14  ; CTL.GLOBAL.HOME.REQUEST.COMPLETED
ORNOT MODE_SEL_MAN  ; MODE.SELECT.MANUAL
OR H3.03  ; MACHINE.CYCLE.STOP
KEEP(011) GLOBAL_HOME_REQUEST  ; GLOBAL.HOME.REQUEST
; rung 1
LD DI_VERT_HOME  ; VERTICAL.AXIS.HOME.PROXIMITY
AND DI_TRANS_HOME  ; TRANSVERSE.AXIS.HOME.PROXIMITY
AND MC_LONG_AXIS_HOME_CMPLT  ; MC.LONG.AXIS.HOMING.COMPLETED
AND DI_LONG_AXIS_HOME_SENS  ; DI.LONG.AXIS.HOME.SENSOR
OUT W0.14  ; CTL.GLOBAL.HOME.REQUEST.COMPLETED
; rung 2
LD GLOBAL_HOME_REQUEST  ; GLOBAL.HOME.REQUEST
ANDNOT DI_VERT_HOME  ; VERTICAL.AXIS.HOME.PROXIMITY
ANDNOT H3.03  ; MACHINE.CYCLE.STOP
OUT W0.13  ; GLOBAL.HOME.REQUEST.HOME.VERTICAL
; rung 3
LD GLOBAL_HOME_REQUEST  ; GLOBAL.HOME.REQUEST
ANDNOT W0.13  ; GLOBAL.HOME.REQUEST.HOME.VERTICAL
ANDNOT DI_TRANS_HOME  ; TRANSVERSE.AXIS.HOME.PROXIMITY
ANDNOT H3.03  ; MACHINE.CYCLE.STOP
OUT W0.12  ; GLOBAL.HOME.REQUEST.HOME.TRANSVERSE
; rung 4
LD GLOBAL_HOME_REQUEST  ; GLOBAL.HOME.REQUEST
ANDNOT W0.12  ; GLOBAL.HOME.REQUEST.HOME.TRANSVERSE
ANDNOT W0.13  ; GLOBAL.HOME.REQUEST.HOME.VERTICAL
ANDNOT DI_LONG_AXIS_HOME_SENS  ; DI.LONG.AXIS.HOME.SENSOR
ANDNOT H3.03  ; MACHINE.CYCLE.STOP
OUT W5.00  ; GLOBAL.HOME.REQUEST.HOME.LONG.TRAVEL
; rung 5
LD DI_LONG_AXIS_HOME_SENS  ; DI.LONG.AXIS.HOME.SENSOR
AND DI_VERT_HOME  ; VERTICAL.AXIS.HOME.PROXIMITY
AND DI_TRANS_HOME  ; TRANSVERSE.AXIS.HOME.PROXIMITY
LD GLOBAL_HOME_REQUEST  ; GLOBAL.HOME.REQUEST
AND P_0_2s
ORLD
OUT W130.00  ; OI.ALL.HOME.INDICATOR

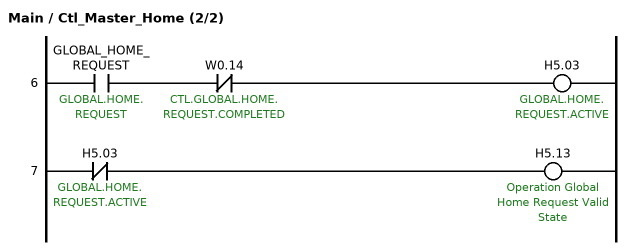
; rung 6
LD GLOBAL_HOME_REQUEST  ; GLOBAL.HOME.REQUEST
ANDNOT W0.14  ; CTL.GLOBAL.HOME.REQUEST.COMPLETED
OUT H5.03  ; GLOBAL.HOME.REQUEST.ACTIVE
; rung 7
LDNOT H5.03  ; GLOBAL.HOME.REQUEST.ACTIVE
OUT H5.13  ; Operation Global Home Request Valid State

### Section Ctl_Long_Axis

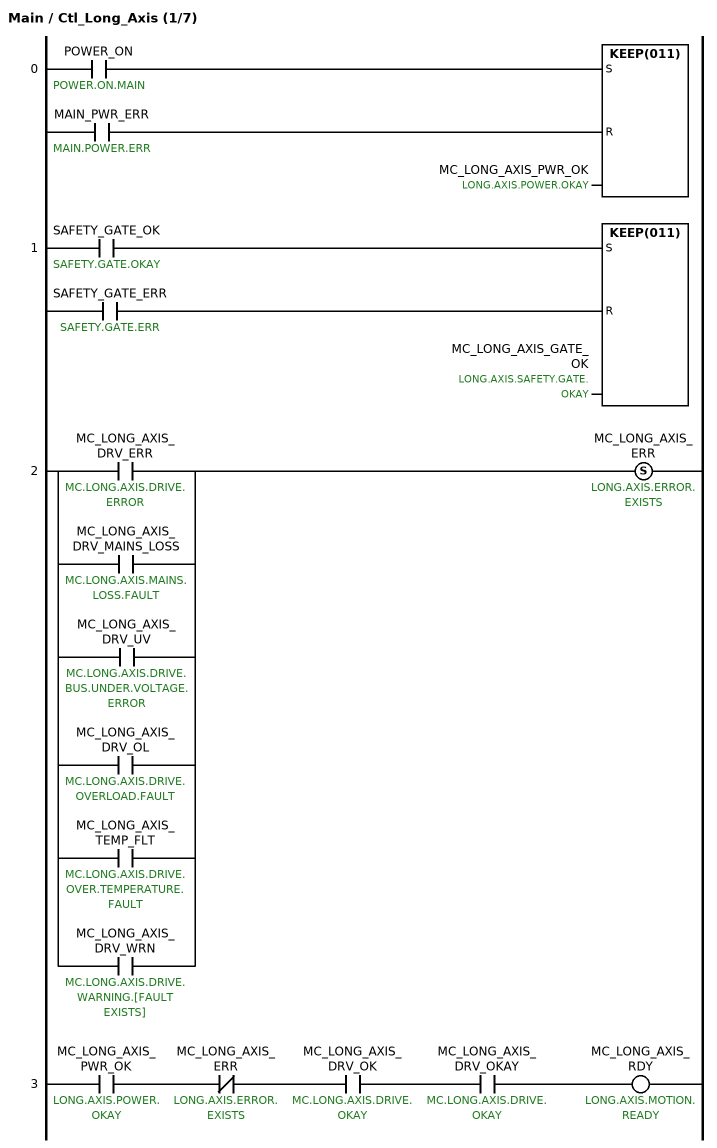
; rung 0
LD POWER_ON  ; POWER.ON.MAIN
LD MAIN_PWR_ERR  ; MAIN.POWER.ERR
KEEP(011) MC_LONG_AXIS_PWR_OK  ; LONG.AXIS.POWER.OKAY
; rung 1
LD SAFETY_GATE_OK  ; SAFETY.GATE.OKAY
LD SAFETY_GATE_ERR  ; SAFETY.GATE.ERR
KEEP(011) MC_LONG_AXIS_GATE_OK  ; LONG.AXIS.SAFETY.GATE.OKAY
; rung 2
LD MC_LONG_AXIS_DRV_ERR  ; MC.LONG.AXIS.DRIVE.ERROR
OR MC_LONG_AXIS_DRV_MAINS_LOSS  ; MC.LONG.AXIS.MAINS.LOSS.FAULT
OR MC_LONG_AXIS_DRV_UV  ; MC.LONG.AXIS.DRIVE.BUS.UNDER.VOLTAGE.ERROR
OR MC_LONG_AXIS_DRV_OL  ; MC.LONG.AXIS.DRIVE.OVERLOAD.FAULT
OR MC_LONG_AXIS_TEMP_FLT  ; MC.LONG.AXIS.DRIVE.OVER.TEMPERATURE.FAULT
OR MC_LONG_AXIS_DRV_WRN  ; MC.LONG.AXIS.DRIVE.WARNING.[FAULT EXISTS]
SET MC_LONG_AXIS_ERR  ; LONG.AXIS.ERROR.EXISTS
; rung 3
LD MC_LONG_AXIS_PWR_OK  ; LONG.AXIS.POWER.OKAY
ANDNOT MC_LONG_AXIS_ERR  ; LONG.AXIS.ERROR.EXISTS
AND MC_LONG_AXIS_DRV_OK  ; MC.LONG.AXIS.DRIVE.OKAY
AND MC_LONG_AXIS_DRV_OKAY  ; MC.LONG.AXIS.DRIVE.OKAY
OUT MC_LONG_AXIS_RDY  ; LONG.AXIS.MOTION.READY

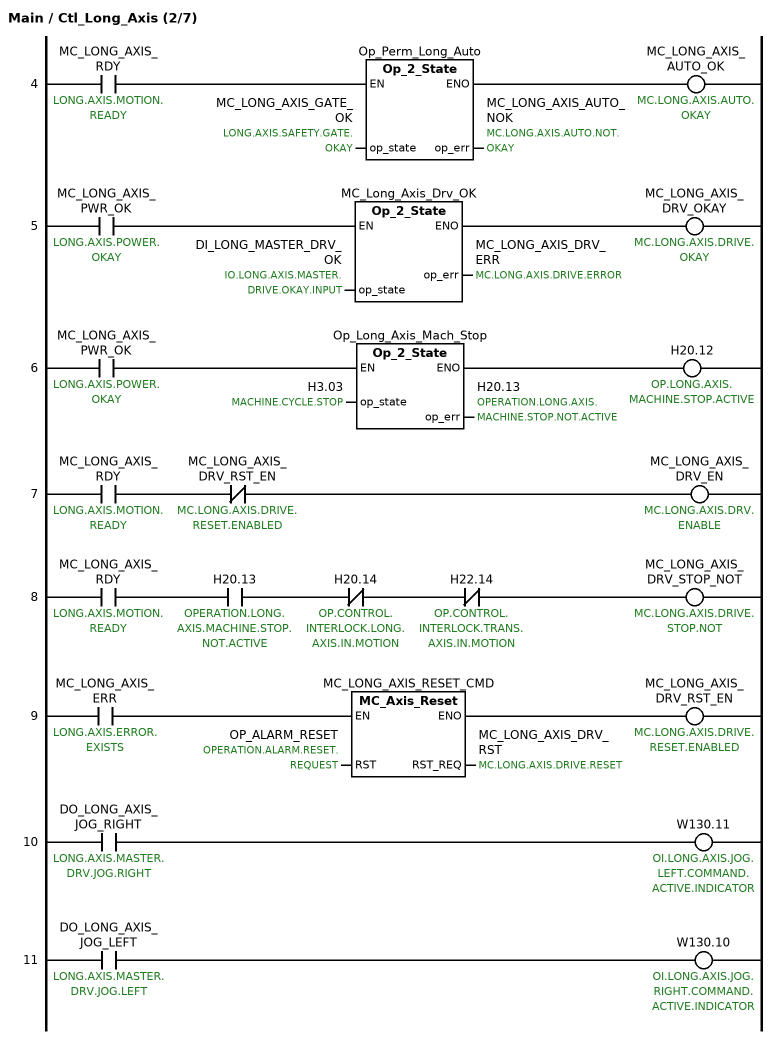
; rung 4
LD MC_LONG_AXIS_RDY  ; LONG.AXIS.MOTION.READY
CALL Op_Perm_Long_Auto : Op_2_State (op_state := MC_LONG_AXIS_GATE_OK, op_err => MC_LONG_AXIS_AUTO_NOK)  ; LONG.AXIS.SAFETY.GATE.OKAY, MC.LONG.AXIS.AUTO.NOT.OKAY
OUT MC_LONG_AXIS_AUTO_OK  ; MC.LONG.AXIS.AUTO.OKAY
; rung 5
LD MC_LONG_AXIS_PWR_OK  ; LONG.AXIS.POWER.OKAY
CALL MC_Long_Axis_Drv_OK : Op_2_State (op_state := DI_LONG_MASTER_DRV_OK, op_err => MC_LONG_AXIS_DRV_ERR)  ; IO.LONG.AXIS.MASTER.DRIVE.OKAY.INPUT, MC.LONG.AXIS.DRIVE.ERROR
OUT MC_LONG_AXIS_DRV_OKAY  ; MC.LONG.AXIS.DRIVE.OKAY
; rung 6
LD MC_LONG_AXIS_PWR_OK  ; LONG.AXIS.POWER.OKAY
CALL Op_Long_Axis_Mach_Stop : Op_2_State (op_state := H3.03, op_err => H20.13)  ; MACHINE.CYCLE.STOP, OPERATION.LONG.AXIS.MACHINE.STOP.NOT.ACTIVE
OUT H20.12  ; OP.LONG.AXIS.MACHINE.STOP.ACTIVE
; rung 7
LD MC_LONG_AXIS_RDY  ; LONG.AXIS.MOTION.READY
ANDNOT MC_LONG_AXIS_DRV_RST_EN  ; MC.LONG.AXIS.DRIVE.RESET.ENABLED
OUT MC_LONG_AXIS_DRV_EN  ; MC.LONG.AXIS.DRV.ENABLE
; rung 8
LD MC_LONG_AXIS_RDY  ; LONG.AXIS.MOTION.READY
AND H20.13  ; OPERATION.LONG.AXIS.MACHINE.STOP.NOT.ACTIVE
ANDNOT H20.14  ; OP.CONTROL.INTERLOCK.LONG.AXIS.IN.MOTION
ANDNOT H22.14  ; OP.CONTROL.INTERLOCK.TRANS.AXIS.IN.MOTION
OUT MC_LONG_AXIS_DRV_STOP_NOT  ; MC.LONG.AXIS.DRIVE.STOP.NOT
; rung 9
LD MC_LONG_AXIS_ERR  ; LONG.AXIS.ERROR.EXISTS
CALL MC_LONG_AXIS_RESET_CMD : MC_Axis_Reset (RST := OP_ALARM_RESET, RST_REQ => MC_LONG_AXIS_DRV_RST)  ; OPERATION.ALARM.RESET.REQUEST, MC.LONG.AXIS.DRIVE.RESET
OUT MC_LONG_AXIS_DRV_RST_EN  ; MC.LONG.AXIS.DRIVE.RESET.ENABLED
; rung 10
LD DO_LONG_AXIS_JOG_RIGHT  ; LONG.AXIS.MASTER.DRV.JOG.RIGHT
OUT W130.11  ; OI.LONG.AXIS.JOG.LEFT.COMMAND.ACTIVE.INDICATOR
; rung 11
LD DO_LONG_AXIS_JOG_LEFT  ; LONG.AXIS.MASTER.DRV.JOG.LEFT
OUT W130.10  ; OI.LONG.AXIS.JOG.RIGHT.COMMAND.ACTIVE.INDICATOR

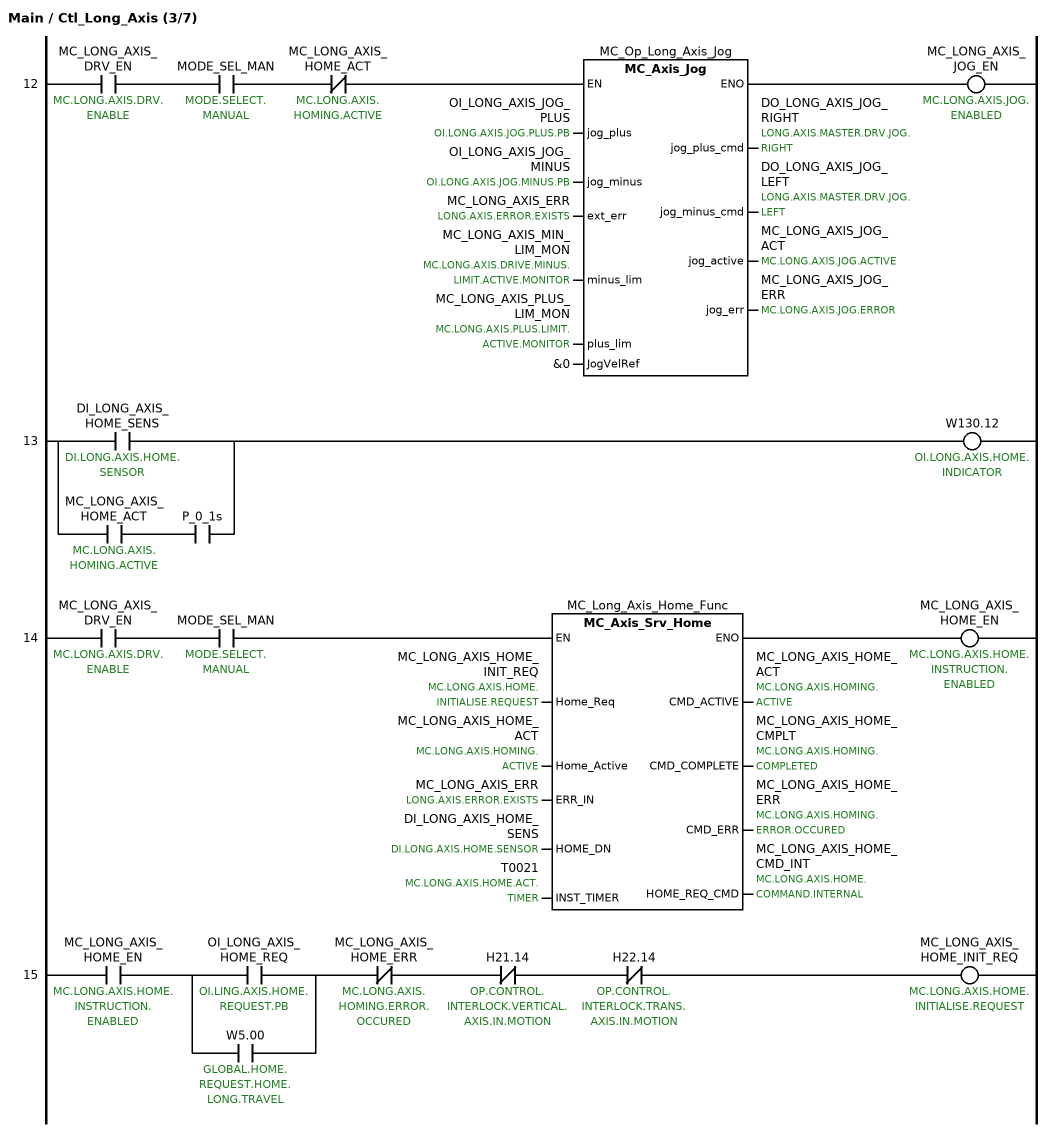
; rung 12
LD MC_LONG_AXIS_DRV_EN  ; MC.LONG.AXIS.DRV.ENABLE
AND MODE_SEL_MAN  ; MODE.SELECT.MANUAL
ANDNOT MC_LONG_AXIS_HOME_ACT  ; MC.LONG.AXIS.HOMING.ACTIVE
CALL MC_Op_Long_Axis_Jog : MC_Axis_Jog (jog_plus := OI_LONG_AXIS_JOG_PLUS, jog_minus := OI_LONG_AXIS_JOG_MINUS, ext_err := MC_LONG_AXIS_ERR, minus_lim := MC_LONG_AXIS_MIN_LIM_MON, plus_lim := MC_LONG_AXIS_PLUS_LIM_MON, JogVelRef := &0, jog_plus_cmd => DO_LONG_AXIS_JOG_RIGHT, jog_minus_cmd => DO_LONG_AXIS_JOG_LEFT, jog_active => MC_LONG_AXIS_JOG_ACT, jog_err => MC_LONG_AXIS_JOG_ERR)  ; OI.LONG.AXIS.JOG.PLUS.PB, OI.LONG.AXIS.JOG.MINUS.PB, LONG.AXIS.ERROR.EXISTS, MC.LONG.AXIS.DRIVE.MINUS.LIMIT.ACTIVE.MONITOR, MC.LONG.AXIS.PLUS.LIMIT.ACTIVE.MONITOR, LONG.AXIS.MASTER.DRV.JOG.RIGHT, LONG.AXIS.MASTER.DRV.JOG.LEFT, MC.LONG.AXIS.JOG.ACTIVE, MC.LONG.AXIS.JOG.ERROR
OUT MC_LONG_AXIS_JOG_EN  ; MC.LONG.AXIS.JOG.ENABLED
; rung 13
LD DI_LONG_AXIS_HOME_SENS  ; DI.LONG.AXIS.HOME.SENSOR
LD MC_LONG_AXIS_HOME_ACT  ; MC.LONG.AXIS.HOMING.ACTIVE
AND P_0_1s
ORLD
OUT W130.12  ; OI.LONG.AXIS.HOME.INDICATOR
; rung 14
LD MC_LONG_AXIS_DRV_EN  ; MC.LONG.AXIS.DRV.ENABLE
AND MODE_SEL_MAN  ; MODE.SELECT.MANUAL
CALL MC_Long_Axis_Home_Func : MC_Axis_Srv_Home (Home_Req := MC_LONG_AXIS_HOME_INIT_REQ, Home_Active := MC_LONG_AXIS_HOME_ACT, ERR_IN := MC_LONG_AXIS_ERR, HOME_DN := DI_LONG_AXIS_HOME_SENS, INST_TIMER := T0021, CMD_ACTIVE => MC_LONG_AXIS_HOME_ACT, CMD_COMPLETE => MC_LONG_AXIS_HOME_CMPLT, CMD_ERR => MC_LONG_AXIS_HOME_ERR, HOME_REQ_CMD => MC_LONG_AXIS_HOME_CMD_INT)  ; MC.LONG.AXIS.HOME.INITIALISE.REQUEST, MC.LONG.AXIS.HOMING.ACTIVE, LONG.AXIS.ERROR.EXISTS, DI.LONG.AXIS.HOME.SENSOR, MC.LONG.AXIS.HOME.ACT.TIMER, MC.LONG.AXIS.HOMING.COMPLETED, MC.LONG.AXIS.HOMING.ERROR.OCCURED, MC.LONG.AXIS.HOME.COMMAND.INTERNAL
OUT MC_LONG_AXIS_HOME_EN  ; MC.LONG.AXIS.HOME.INSTRUCTION.ENABLED
; rung 15
LD MC_LONG_AXIS_HOME_EN  ; MC.LONG.AXIS.HOME.INSTRUCTION.ENABLED
LD OI_LONG_AXIS_HOME_REQ  ; OI.LING.AXIS.HOME.REQUEST.PB
OR W5.00  ; GLOBAL.HOME.REQUEST.HOME.LONG.TRAVEL
ANDLD
ANDNOT MC_LONG_AXIS_HOME_ERR  ; MC.LONG.AXIS.HOMING.ERROR.OCCURED
ANDNOT H21.14  ; OP.CONTROL.INTERLOCK.VERTICAL.AXIS.IN.MOTION
ANDNOT H22.14  ; OP.CONTROL.INTERLOCK.TRANS.AXIS.IN.MOTION
OUT MC_LONG_AXIS_HOME_INIT_REQ  ; MC.LONG.AXIS.HOME.INITIALISE.REQUEST

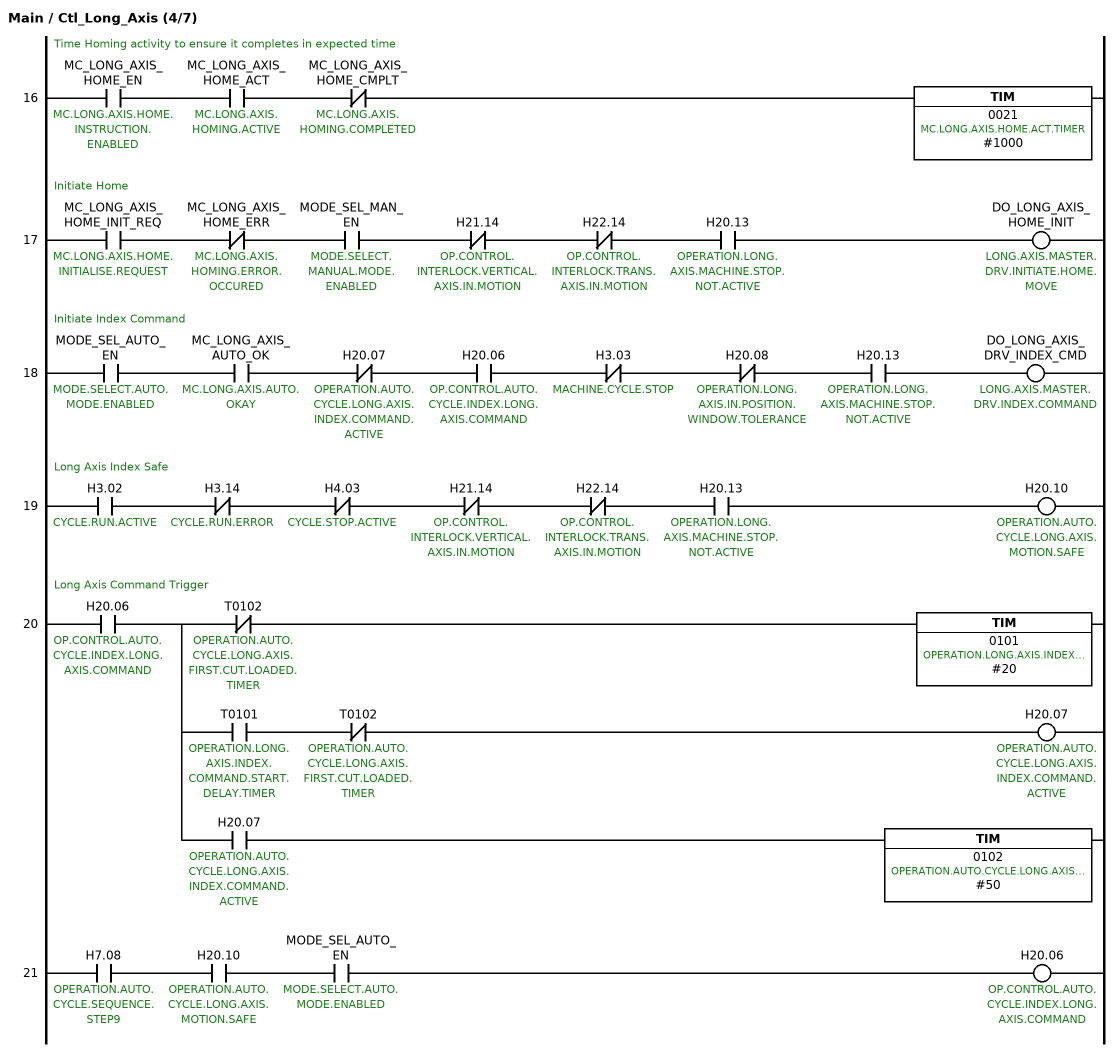
; rung 16: Time Homing activity to ensure it completes in expected time
LD MC_LONG_AXIS_HOME_EN  ; MC.LONG.AXIS.HOME.INSTRUCTION.ENABLED
AND MC_LONG_AXIS_HOME_ACT  ; MC.LONG.AXIS.HOMING.ACTIVE
ANDNOT MC_LONG_AXIS_HOME_CMPLT  ; MC.LONG.AXIS.HOMING.COMPLETED
TIM 0021 #1000  ; MC.LONG.AXIS.HOME.ACT.TIMER
; rung 17: Initiate Home
LD MC_LONG_AXIS_HOME_INIT_REQ  ; MC.LONG.AXIS.HOME.INITIALISE.REQUEST
ANDNOT MC_LONG_AXIS_HOME_ERR  ; MC.LONG.AXIS.HOMING.ERROR.OCCURED
AND MODE_SEL_MAN_EN  ; MODE.SELECT.MANUAL.MODE.ENABLED
ANDNOT H21.14  ; OP.CONTROL.INTERLOCK.VERTICAL.AXIS.IN.MOTION
ANDNOT H22.14  ; OP.CONTROL.INTERLOCK.TRANS.AXIS.IN.MOTION
AND H20.13  ; OPERATION.LONG.AXIS.MACHINE.STOP.NOT.ACTIVE
OUT DO_LONG_AXIS_HOME_INIT  ; LONG.AXIS.MASTER.DRV.INITIATE.HOME.MOVE
; rung 18: Initiate Index Command
LD MODE_SEL_AUTO_EN  ; MODE.SELECT.AUTO.MODE.ENABLED
AND MC_LONG_AXIS_AUTO_OK  ; MC.LONG.AXIS.AUTO.OKAY
ANDNOT H20.07  ; OPERATION.AUTO.CYCLE.LONG.AXIS.INDEX.COMMAND.ACTIVE
AND H20.06  ; OP.CONTROL.AUTO.CYCLE.INDEX.LONG.AXIS.COMMAND
ANDNOT H3.03  ; MACHINE.CYCLE.STOP
ANDNOT H20.08  ; OPERATION.LONG.AXIS.IN.POSITION.WINDOW.TOLERANCE
AND H20.13  ; OPERATION.LONG.AXIS.MACHINE.STOP.NOT.ACTIVE
OUT DO_LONG_AXIS_DRV_INDEX_CMD  ; LONG.AXIS.MASTER.DRV.INDEX.COMMAND
; rung 19: Long Axis Index Safe
LD H3.02  ; CYCLE.RUN.ACTIVE
ANDNOT H3.14  ; CYCLE.RUN.ERROR
ANDNOT H4.03  ; CYCLE.STOP.ACTIVE
ANDNOT H21.14  ; OP.CONTROL.INTERLOCK.VERTICAL.AXIS.IN.MOTION
ANDNOT H22.14  ; OP.CONTROL.INTERLOCK.TRANS.AXIS.IN.MOTION
AND H20.13  ; OPERATION.LONG.AXIS.MACHINE.STOP.NOT.ACTIVE
OUT H20.10  ; OPERATION.AUTO.CYCLE.LONG.AXIS.MOTION.SAFE
; rung 20: Long Axis Command Trigger
LD H20.06  ; OP.CONTROL.AUTO.CYCLE.INDEX.LONG.AXIS.COMMAND
OUT TR0
ANDNOT T0102  ; OPERATION.AUTO.CYCLE.LONG.AXIS.FIRST.CUT.LOADED.TIMER
TIM 0101 #20  ; OPERATION.LONG.AXIS.INDEX.COMMAND.START.DELAY.TIMER
LD TR0
AND T0101  ; OPERATION.LONG.AXIS.INDEX.COMMAND.START.DELAY.TIMER
ANDNOT T0102  ; OPERATION.AUTO.CYCLE.LONG.AXIS.FIRST.CUT.LOADED.TIMER
OUT H20.07  ; OPERATION.AUTO.CYCLE.LONG.AXIS.INDEX.COMMAND.ACTIVE
LD TR0
AND H20.07  ; OPERATION.AUTO.CYCLE.LONG.AXIS.INDEX.COMMAND.ACTIVE
TIM 0102 #50  ; OPERATION.AUTO.CYCLE.LONG.AXIS.FIRST.CUT.LOADED.TIMER
; rung 21
LD H7.08  ; OPERATION.AUTO.CYCLE.SEQUENCE.STEP9
AND H20.10  ; OPERATION.AUTO.CYCLE.LONG.AXIS.MOTION.SAFE
AND MODE_SEL_AUTO_EN  ; MODE.SELECT.AUTO.MODE.ENABLED
OUT H20.06  ; OP.CONTROL.AUTO.CYCLE.INDEX.LONG.AXIS.COMMAND

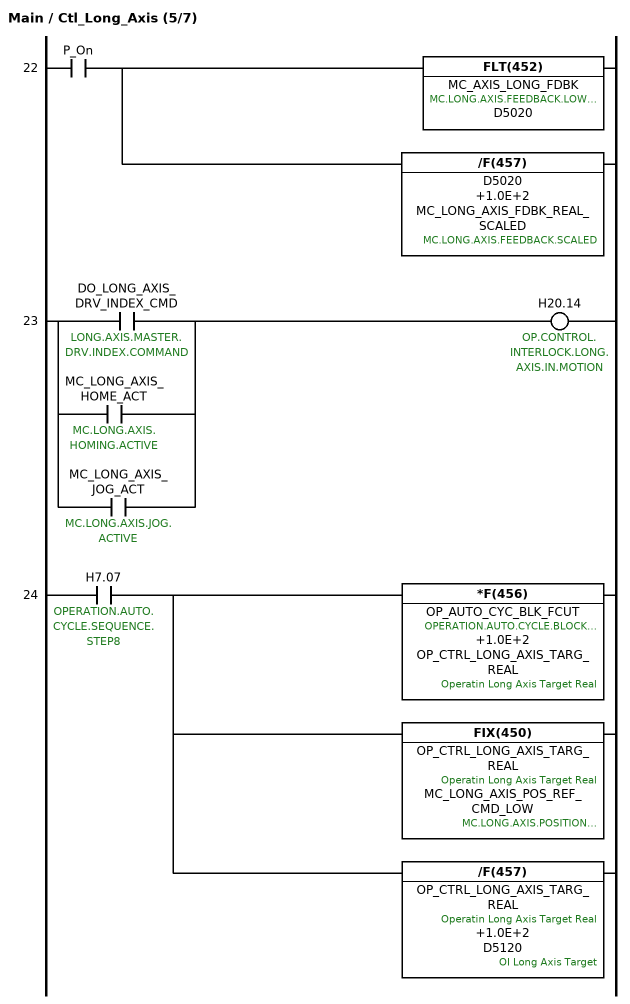
; rung 22
LD P_On
FLT(452) MC_AXIS_LONG_FDBK D5020  ; MC.LONG.AXIS.FEEDBACK.LOW.WORD
/F(457) D5020 +1.0E+2 MC_LONG_AXIS_FDBK_REAL_SCALED  ; MC.LONG.AXIS.FEEDBACK.SCALED
; rung 23
LD DO_LONG_AXIS_DRV_INDEX_CMD  ; LONG.AXIS.MASTER.DRV.INDEX.COMMAND
OR MC_LONG_AXIS_HOME_ACT  ; MC.LONG.AXIS.HOMING.ACTIVE
OR MC_LONG_AXIS_JOG_ACT  ; MC.LONG.AXIS.JOG.ACTIVE
OUT H20.14  ; OP.CONTROL.INTERLOCK.LONG.AXIS.IN.MOTION
; rung 24
LD H7.07  ; OPERATION.AUTO.CYCLE.SEQUENCE.STEP8
*F(456) OP_AUTO_CYC_BLK_FCUT +1.0E+2 OP_CTRL_LONG_AXIS_TARG_REAL  ; OPERATION.AUTO.CYCLE.BLOCK.FIRST.CUT.WORKING, Operatin Long Axis Target Real
FIX(450) OP_CTRL_LONG_AXIS_TARG_REAL MC_LONG_AXIS_POS_REF_CMD_LOW  ; Operatin Long Axis Target Real, MC.LONG.AXIS.POSITION.REFERENCE.COMMAND.VALUE.LOW.WORD
/F(457) OP_CTRL_LONG_AXIS_TARG_REAL +1.0E+2 D5120  ; Operatin Long Axis Target Real, OI Long Axis Target

